// TIA Portal V19 export
FUNCTION_BLOCK "FDevice_Sinamics_FB"   // FB49, F_LAD
// stored: Access Published
   VAR_INPUT
      Tlg30_IN { ExternalAccessible := 'False'; ExternalVisible := 'False'; ExternalWritable := 'False'} : "udt_LDrvSafe_typeSinaSTlg30Status";
      Estop : Bool;
      Two_Hand_CMD : Bool;   // Safe Motion Command
      Door_SafeStop : Bool;   // Safe Stop from Doors
      CtrlSafe : Bool;   // Movement is Required
      EnableSOS : Bool;   // Enable SOS
      EnableSS1 : Bool;   // EnableSS1
      Reset : Bool;
      StoppingTime : Time := T#2s;   // Movement stopping time
   END_VAR
   VAR_OUTPUT
      Tlg30_OUT { ExternalAccessible := 'False'; ExternalVisible := 'False'; ExternalWritable := 'False'} : "udt_LDrvSafe_typeSinaSTlg30Control";
      SftyFault : Bool;   // Drive has a Safety Fault Active
   END_VAR
   VAR_IN_OUT
      DSI : "udt_DeviceSafetyInterface";   // Device Safety Interface
   END_VAR
   VAR
      DriveT30_Ctrl : "LDrvSafe_SinaSTlg30Control";   // Ctrl
      DriveT30_Sts : "LDrvSafe_SinaSTlg30Status";   // Sts
      T_StopDelay : TOF;
      T_StoDelay : TOF;
      T_SlsDelay : TOF;
   END_VAR
   VAR_TEMP
      S_ON : Bool;
      STO : Bool;
   END_VAR
BEGIN

REGION Network 1: Safety Enable
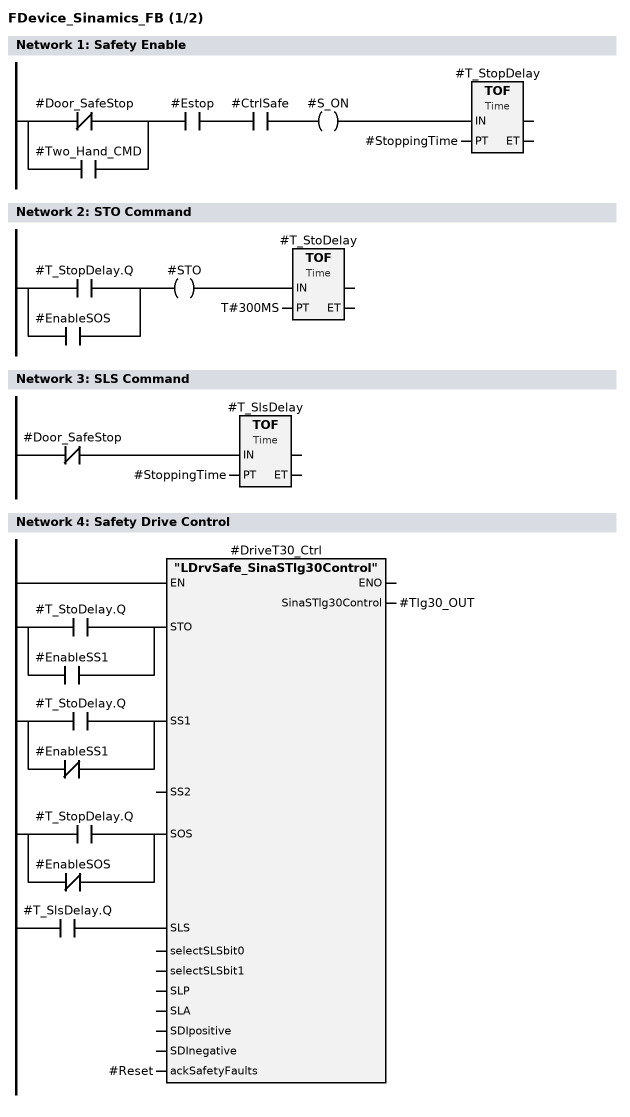
   RUNG wire#powerrail
      I_Contact( #Door_SafeStop )
      wire#w1
      Contact( #Estop )
      Contact( #CtrlSafe )
      Coil( #S_ON )
      { S7_Templates := "[time_type := Time, codedbool_type := DInt]" } #T_StopDelay.TOF(pt := #StoppingTime, et =>)
   END_RUNG
   RUNG wire#powerrail
      Contact( #Two_Hand_CMD )
   END_RUNG wire#w1
   // the same network as SCL:
   #S_ON := (NOT #Door_SafeStop OR #Two_Hand_CMD) AND #Estop AND #CtrlSafe;
   #T_StopDelay.TOF(IN := #S_ON, PT := #StoppingTime);
END_REGION

REGION Network 2: STO Command
   RUNG wire#powerrail
      Contact( #T_StopDelay.Q )
      wire#w1
      Coil( #STO )
      { S7_Templates := "[time_type := Time, codedbool_type := DInt]" } #T_StoDelay.TOF(pt := T#300MS, et =>)
   END_RUNG
   RUNG wire#powerrail
      Contact( #EnableSOS )
   END_RUNG wire#w1
   // the same network as SCL:
   #STO := #T_StopDelay.Q OR #EnableSOS;
   #T_StoDelay.TOF(IN := #STO, PT := T#300MS);
END_REGION

REGION Network 3: SLS Command
   RUNG wire#powerrail
      I_Contact( #Door_SafeStop )
      { S7_Templates := "[time_type := Time, codedbool_type := DInt]" } #T_SlsDelay.TOF(pt := #StoppingTime, et =>)
   END_RUNG
   // the same network as SCL:
   #T_SlsDelay.TOF(IN := NOT #Door_SafeStop, PT := #StoppingTime);
END_REGION

REGION Network 4: Safety Drive Control
   RUNG wire#powerrail
      #DriveT30_Ctrl(STO := wire#w1, SS1 := wire#w2, SOS := wire#w3, SLS := wire#w4, SS2 :=, selectSLSbit0 :=, selectSLSbit1 :=, SLP :=, SLA :=, SDIpositive :=, SDInegative :=, ackSafetyFaults := #Reset, SinaSTlg30Control => #Tlg30_OUT)
   END_RUNG
   RUNG wire#powerrail
      Contact( #T_StoDelay.Q )
   END_RUNG wire#w1
   RUNG wire#powerrail
      Contact( #EnableSS1 )
   END_RUNG wire#w1
   RUNG wire#powerrail
      Contact( #T_StoDelay.Q )
   END_RUNG wire#w2
   RUNG wire#powerrail
      I_Contact( #EnableSS1 )
   END_RUNG wire#w2
   RUNG wire#powerrail
      Contact( #T_StopDelay.Q )
   END_RUNG wire#w3
   RUNG wire#powerrail
      I_Contact( #EnableSOS )
   END_RUNG wire#w3
   RUNG wire#powerrail
      Contact( #T_SlsDelay.Q )
   END_RUNG wire#w4
   // the same network as SCL:
   #DriveT30_Ctrl(STO := #T_StoDelay.Q OR #EnableSS1,   // "LDrvSafe_SinaSTlg30Control"
                  SS1 := #T_StoDelay.Q OR NOT #EnableSS1,
                  SOS := #T_StopDelay.Q OR NOT #EnableSOS,
                  SLS := #T_SlsDelay.Q,
                  ackSafetyFaults := #Reset,
                  SinaSTlg30Control => #Tlg30_OUT);
END_REGION

REGION Network 5: Safety Drive Status
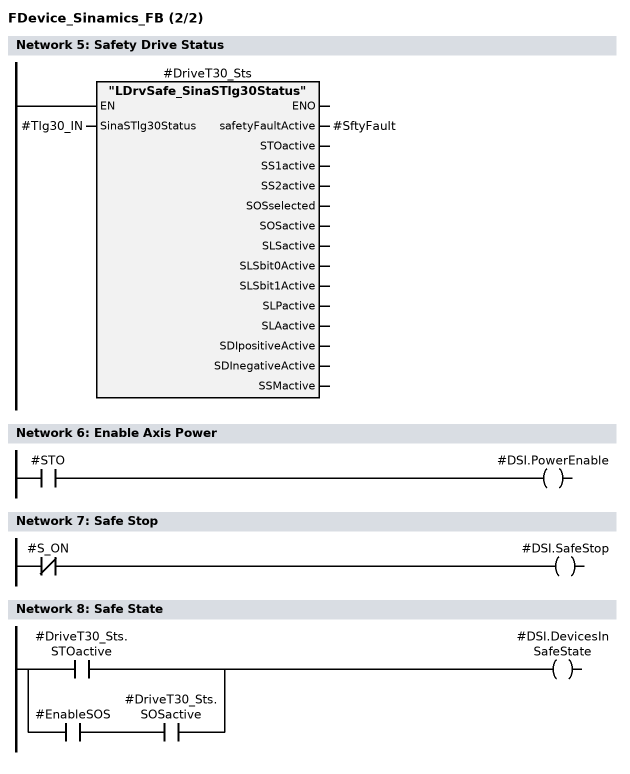
   RUNG wire#powerrail
      #DriveT30_Sts(SinaSTlg30Status := #Tlg30_IN, safetyFaultActive => #SftyFault, STOactive =>, SS1active =>, SS2active =>, SOSselected =>, SOSactive =>, SLSactive =>, SLSbit0Active =>, SLSbit1Active =>, SLPactive =>, SLAactive =>, SDIpositiveActive =>, SDInegativeActive =>, SSMactive =>)
   END_RUNG
   // the same network as SCL:
   #DriveT30_Sts(SinaSTlg30Status := #Tlg30_IN, safetyFaultActive => #SftyFault);   // "LDrvSafe_SinaSTlg30Status"
END_REGION

REGION Network 6: Enable Axis Power
   RUNG wire#powerrail
      Contact( #STO )
      Coil( #DSI.PowerEnable )
   END_RUNG
   // the same network as SCL:
   #DSI.PowerEnable := #STO;
END_REGION

REGION Network 7: Safe Stop
   RUNG wire#powerrail
      I_Contact( #S_ON )
      Coil( #DSI.SafeStop )
   END_RUNG
   // the same network as SCL:
   #DSI.SafeStop := NOT #S_ON;
END_REGION

REGION Network 8: Safe State
   RUNG wire#powerrail
      Contact( #DriveT30_Sts.STOactive )
      wire#w1
      Coil( #DSI.DevicesInSafeState )
   END_RUNG
   RUNG wire#powerrail
      Contact( #EnableSOS )
      Contact( #DriveT30_Sts.SOSactive )
   END_RUNG wire#w1
   // the same network as SCL:
   #DSI.DevicesInSafeState := #DriveT30_Sts.STOactive OR (#EnableSOS AND #DriveT30_Sts.SOSactive);
END_REGION
END_FUNCTION_BLOCK
